{attribute 'GeneratedUsingTerminal: EL4004-0000-0020'}
{attribute addProperty BoxType "EL4004-0000-0020"}
{attribute addProperty Id "AO_Outputs_Channel_1AT %Q*AO_Outputs_Channel_BA7EBB7C2AO_Outputs_Channel_2AT %Q*AO_Outputs_Channel_BA7EBB7C2AO_Outputs_Channel_3AT %Q*AO_Outputs_Channel_BA7EBB7C2AO_Outputs_Channel_4AT %Q*AO_Outputs_Channel_BA7EBB7C2WcStateAT %I*WcState_0B2B16F91InfoDataAT %I*InfoData_32EB74EA10"}
{attribute addProperty CRC "3534211511"}
{attribute addProperty Size "19"}
TYPE EL4004_D2A7C9B7 :
STRUCT
	{attribute addProperty Name "AO_Outputs_Channel_1"}
	AO_Outputs_Channel_1 : AO_Outputs_Channel_BA7EBB7C;
	{attribute addProperty Name "AO_Outputs_Channel_2"}
	AO_Outputs_Channel_2 : AO_Outputs_Channel_BA7EBB7C;
	{attribute addProperty Name "AO_Outputs_Channel_3"}
	AO_Outputs_Channel_3 : AO_Outputs_Channel_BA7EBB7C;
	{attribute addProperty Name "AO_Outputs_Channel_4"}
	AO_Outputs_Channel_4 : AO_Outputs_Channel_BA7EBB7C;
	{attribute addProperty Name "WcState"}
	WcState : TcoIoBeckhoff.WcState_0B2B16F9;
	{attribute addProperty Name "InfoData"}
	InfoData : InfoData_32EB74EA;
END_STRUCT
END_TYPE

(* stored: Version 1.2.0.0, ProductVersion 3.1.4024.9
   DUT EL4004_D2A7C9B7: Id {5b9040df-40cc-0742-09f1-fde001838f71} *)
